_CFC_ (* Continuous Function Chart, elements in execution order *)
(* 85% от частоты вращения *)
(* 60% от частоты вращения *)
#0 WORD_TO_REAL(RD_1[0])
#1 DIV(#0, 100)
#2 SCHU_P2_2_M1_OBR <= #1
#3 dost_ton:TON(IN: NOT SCHU_P2_2_M1_OBR_ERROR, PT: t#10s)
#4 SR_DOST_M1:RS(SET: #3.Q, RESET1: SCHU_P2_2_M1_OBR_ERROR)
#5 DIV(SCHU_P2_2_SPEEDMOTOR, 100)
#6 MUL(#5, 60)
#7 fb_M1b30:ISTOK_GT(dost: #4.Q1, x: SCHU_P2_2_M1_OBR, ust: #6, shkal: -, gist: 1)
#8 SCHU_P2_2_M1_B30 <= #7.Xb
#9 DIV(SCHU_P2_2_SPEEDMOTOR, 100)
#10 MUL(#9, 85)
#11 fb_M1_OBRb45:ISTOK_GT(dost: #4.Q1, x: SCHU_P2_2_M1_OBR, ust: #10, shkal: -, gist: 1)
#12 SCHU_P2_2_M1_B45 <= #11.Xb
#13 fb_M1_OBRm0_1:ISTOK_LT(dost: #4.Q1, x: SCHU_P2_2_M1_OBR, ust: 0.1, shkal: -, gist: 1)
#14 SCHU_P2_2_M1_M0_1 <= #13.Xm
#15 fb_M1_OBRbSM:ISTOK_GT(dost: #4.Q1, x: SCHU_P2_2_M1_OBR, ust: SCHU_P2_2_SPEEDMOTOR, shkal: -, gist: 1)
#16 SCHU_P2_2_M1_OBRBSM <= #15.Xb
_END_CFC_
(* the same logic as Structured Text *)
(* 85% от частоты вращения *)
(* 60% от частоты вращения *)
SCHU_P2_2_M1_OBR := WORD_TO_REAL(RD_1[0]) / 100;
dost_ton(IN := NOT SCHU_P2_2_M1_OBR_ERROR, PT := t#10s);
SR_DOST_M1(SET := dost_ton.Q, RESET1 := SCHU_P2_2_M1_OBR_ERROR);
fb_M1b30(dost := SR_DOST_M1.Q1, x := SCHU_P2_2_M1_OBR, ust := (SCHU_P2_2_SPEEDMOTOR / 100) * 60, gist := 1);
SCHU_P2_2_M1_B30 := fb_M1b30.Xb;
fb_M1_OBRb45(dost := SR_DOST_M1.Q1, x := SCHU_P2_2_M1_OBR, ust := (SCHU_P2_2_SPEEDMOTOR / 100) * 85, gist := 1);
SCHU_P2_2_M1_B45 := fb_M1_OBRb45.Xb;
fb_M1_OBRm0_1(dost := SR_DOST_M1.Q1, x := SCHU_P2_2_M1_OBR, ust := 0.1, gist := 1);
SCHU_P2_2_M1_M0_1 := fb_M1_OBRm0_1.Xm;
fb_M1_OBRbSM(dost := SR_DOST_M1.Q1, x := SCHU_P2_2_M1_OBR, ust := SCHU_P2_2_SPEEDMOTOR, gist := 1);
SCHU_P2_2_M1_OBRBSM := fb_M1_OBRbSM.Xb;
END_PROGRAM

(* POU Input/CI/M2_OB, CFC *)
PROGRAM M2_OB
VAR
	fb_M2_OBRbSM: ISTOK_GT;
	fb_M2b30: ISTOK_GT;
	fb_M2_OBRm0_1: ISTOK_LT;
	fb_M2_OBRb45: ISTOK_GT;
	fb_M2_OBR: ISTOK_ANALOGVH;
	ofset: INT := 0;
	SR_DOST_M2: RS;
	dost_ton_2: TON;
END_VAR
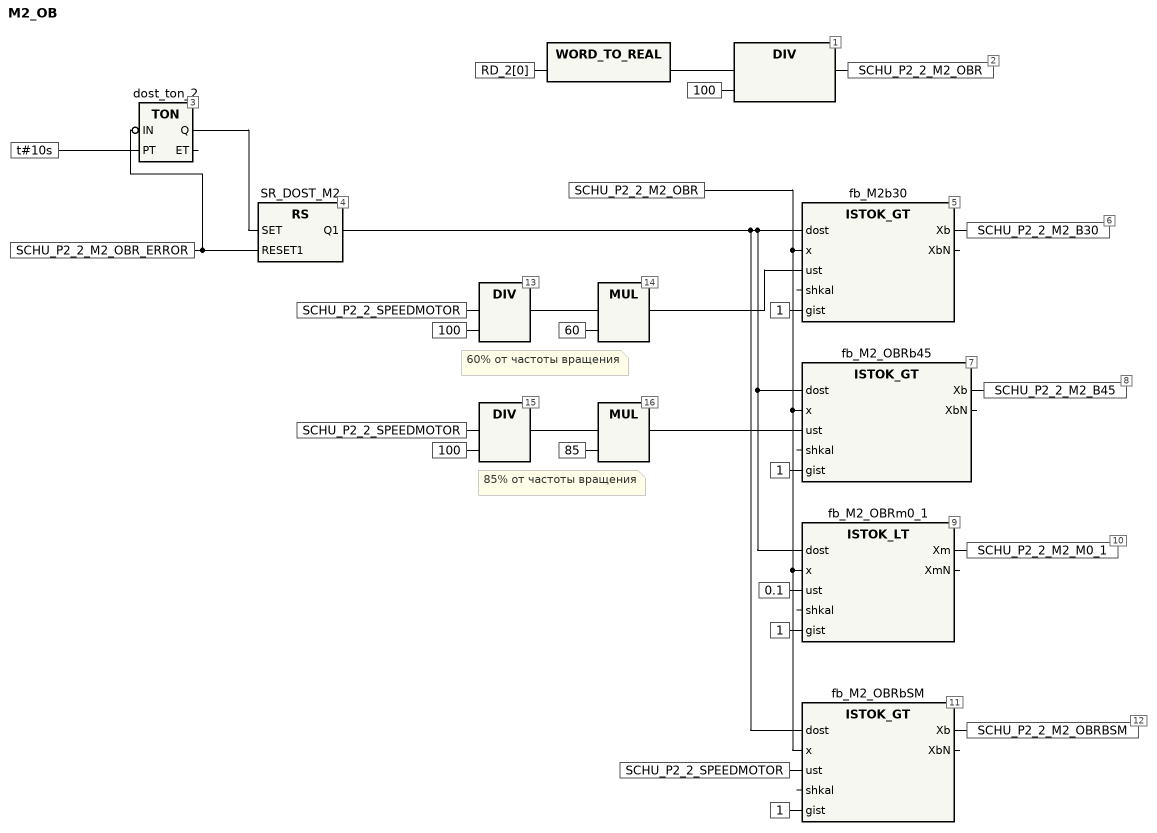
_CFC_ (* Continuous Function Chart, elements in execution order *)
#0 WORD_TO_REAL(RD_2[0])
#1 DIV(#0, 100)
#2 SCHU_P2_2_M2_OBR <= #1
#3 dost_ton_2:TON(IN: NOT SCHU_P2_2_M2_OBR_ERROR, PT: t#10s)
#4 SR_DOST_M2:RS(SET: #3.Q, RESET1: SCHU_P2_2_M2_OBR_ERROR)
#5 fb_M2b30:ISTOK_GT(dost: #4.Q1, x: SCHU_P2_2_M2_OBR, ust: #14, shkal: -, gist: 1)
#6 SCHU_P2_2_M2_B30 <= #5.Xb
#7 fb_M2_OBRb45:ISTOK_GT(dost: #4.Q1, x: SCHU_P2_2_M2_OBR, ust: #16, shkal: -, gist: 1)
#8 SCHU_P2_2_M2_B45 <= #7.Xb
#9 fb_M2_OBRm0_1:ISTOK_LT(dost: #4.Q1, x: SCHU_P2_2_M2_OBR, ust: 0.1, shkal: -, gist: 1)
#10 SCHU_P2_2_M2_M0_1 <= #9.Xm
#11 fb_M2_OBRbSM:ISTOK_GT(dost: #4.Q1, x: SCHU_P2_2_M2_OBR, ust: SCHU_P2_2_SPEEDMOTOR, shkal: -, gist: 1)
#12 SCHU_P2_2_M2_OBRBSM <= #11.Xb
(* 60% от частоты вращения *)
#13 DIV(SCHU_P2_2_SPEEDMOTOR, 100)
#14 MUL(#13, 60)
#15 DIV(SCHU_P2_2_SPEEDMOTOR, 100)
#16 MUL(#15, 85)
(* 85% от частоты вращения *)
_END_CFC_
END_PROGRAM

(* POU Input/AI/UE1_T, CFC *)
PROGRAM UE1_T
VAR
	fb_UE2_T: ISTOK_ANALOGVH;
	ofset: REAL;
	fb_UE2eqUST: ISTOK_EQ;
	fb_UE2_m_UST: ISTOK_LT;
	fb_UE2_b_UST: ISTOK_GT;
	enbleLimit: BOOL;
END_VAR
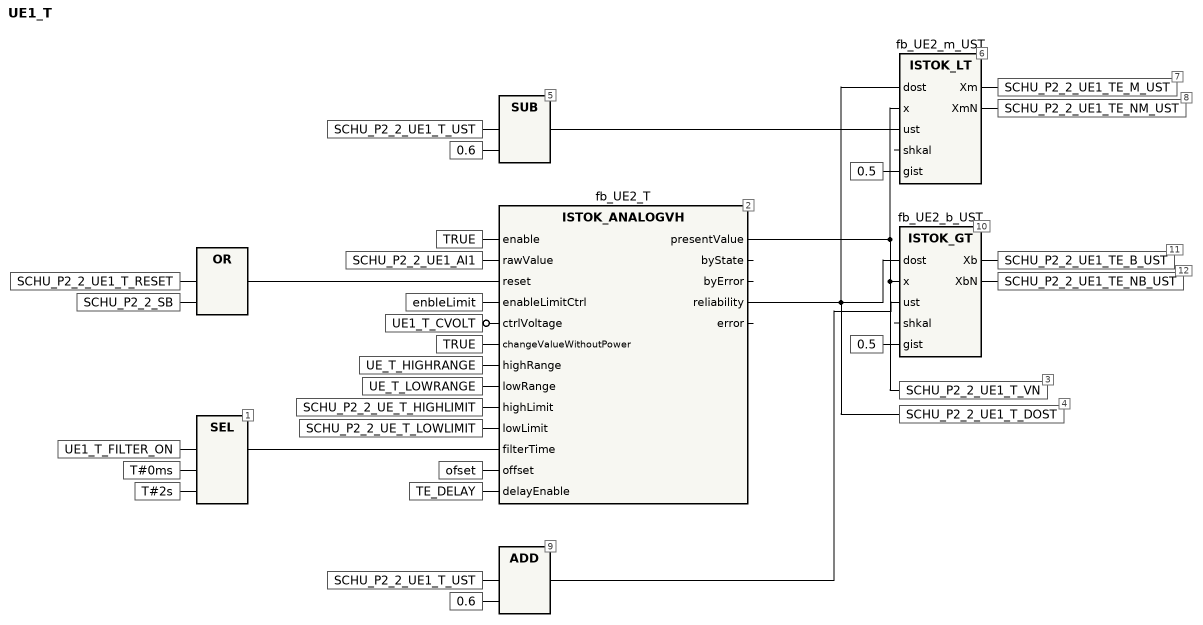
